Fanuc KAREL source: kt00889.KL

-- PROVISIONAL review KL for V770-1; original PC SHA256 f4216a5a5d83b9ecd9c9835330bab15fee24f90de36bb538c76b4df140c3a128
-- Incomplete behavior may be omitted. Consult companion uncertainty JSON. Do not deploy.
PROGRAM KT00889
%NOLOCKGROUP
-- UNRESOLVED_DECL P1 type=000102
-- UNRESOLVED_DECL P2 type=000102
-- UNRESOLVED_DECL OUT type=000101
BEGIN
  -- UNRESOLVED_PC offsets 5-20; opcodes 2E,22,32,35
  -- UNRESOLVED_PC offsets 25-40; opcodes 2E,22,32,35
  -- UNRESOLVED_PC offsets 45-60; opcodes 2E,22,32,35
  -- UNRESOLVED_PC offsets 65-80; opcodes 2E,22,32,35
  -- UNRESOLVED_PC offsets 85-115; opcodes 27,27,49,7E,AD,76,7E,4A
  -- UNRESOLVED_PC offsets 120-124; opcodes 7F
END KT00889
